FUNCTION_BLOCK CmdVentValves (* CAT Function Block Type *)
  (* Standard: 61499-2 *)
  (* Version 0.0, 6/8/2026, Schneider Electric, template *)
  PACKAGE SE.Nereda;
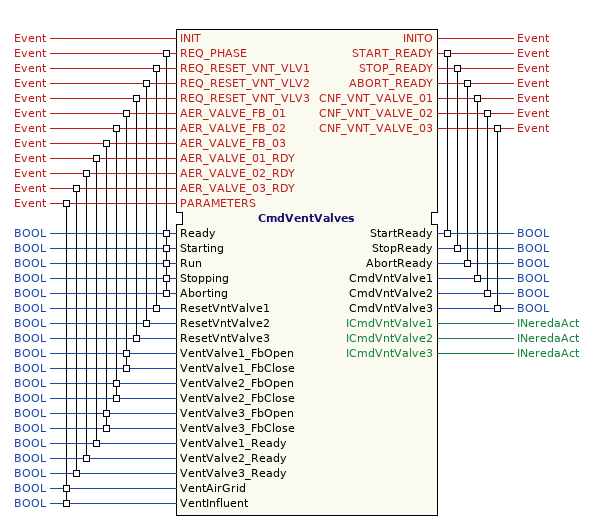
  EVENT_INPUT
    INIT;
    REQ_PHASE WITH Ready, Starting, Run, Stopping, Aborting;
    REQ_RESET_VNT_VLV1 WITH ResetVntValve1;
    REQ_RESET_VNT_VLV2 WITH ResetVntValve2;
    REQ_RESET_VNT_VLV3 WITH ResetVntValve3;
    AER_VALVE_FB_01 WITH VentValve1_FbOpen, VentValve1_FbClose;
    AER_VALVE_FB_02 WITH VentValve2_FbOpen, VentValve2_FbClose;
    AER_VALVE_FB_03 WITH VentValve3_FbOpen, VentValve3_FbClose;
    AER_VALVE_01_RDY WITH VentValve1_Ready;
    AER_VALVE_02_RDY WITH VentValve2_Ready;
    AER_VALVE_03_RDY WITH VentValve3_Ready;
    PARAMETERS WITH VentAirGrid, VentInfluent;
  END_EVENT
  EVENT_OUTPUT
    INITO;
    START_READY WITH StartReady;
    STOP_READY WITH StopReady;
    ABORT_READY WITH AbortReady;
    CNF_VNT_VALVE_01 WITH CmdVntValve1;
    CNF_VNT_VALVE_02 WITH CmdVntValve2;
    CNF_VNT_VALVE_03 WITH CmdVntValve3;
  END_EVENT
  VAR_INPUT
    Ready : BOOL;
    Starting : BOOL;
    Run : BOOL;
    Stopping : BOOL;
    Aborting : BOOL;
    ResetVntValve1 : BOOL;
    ResetVntValve2 : BOOL;
    ResetVntValve3 : BOOL;
    VentValve1_FbOpen : BOOL;
    VentValve1_FbClose : BOOL;
    VentValve2_FbOpen : BOOL;
    VentValve2_FbClose : BOOL;
    VentValve3_FbOpen : BOOL;
    VentValve3_FbClose : BOOL;
    VentValve1_Ready : BOOL;
    VentValve2_Ready : BOOL;
    VentValve3_Ready : BOOL;
    VentAirGrid : BOOL;
    VentInfluent : BOOL;
  END_VAR
  VAR_OUTPUT
    StartReady : BOOL;
    StopReady : BOOL;
    AbortReady : BOOL;
    CmdVntValve1 : BOOL;
    CmdVntValve2 : BOOL;
    CmdVntValve3 : BOOL;
  END_VAR
  PLUGS
    ICmdVntValve1 : INeredaAct;
    ICmdVntValve2 : INeredaAct;
    ICmdVntValve3 : INeredaAct;
  END_PLUGS
  (* 01 - FUNCTIONNAL INPUT INTERFACE *)
  (* 00 - INITIALIZATION *)
  (* 05 - LOGIC *)
  (* 06 - HMI INTERFACE *)
  (* 03 - FIELD INTERFACE *)
  (* 02 - FUNCTIONNAL OUTPUT INTERFACE *)
  (* Command Logic *)
  FBS
    IThis : CmdVentValves_HMI(QI := TRUE);
    CmdAerationValve1 : boolValueChanged;
    CmdAerationValve2 : boolValueChanged;
    FbOpenValve1 : DS_SELECTX_2536758B411A6CE51; {SET_ATTRIBUTE(Configuration.GenericFBType.InterfaceParams, Runtime.Standard#CNTX:=2;CNTY:=1;DI${CNTX,_,CNTY$}:BOOL)}
    FbCloseValve1 : DS_SELECTX_2536758B411A6CE51; {SET_ATTRIBUTE(Configuration.GenericFBType.InterfaceParams, Runtime.Standard#CNTX:=2;CNTY:=1;DI${CNTX,_,CNTY$}:BOOL)}
    FbOpenValve3 : DS_SELECTX_2536758B411A6CE51; {SET_ATTRIBUTE(Configuration.GenericFBType.InterfaceParams, Runtime.Standard#CNTX:=2;CNTY:=1;DI${CNTX,_,CNTY$}:BOOL)}
    FbCloseValve3 : DS_SELECTX_2536758B411A6CE51; {SET_ATTRIBUTE(Configuration.GenericFBType.InterfaceParams, Runtime.Standard#CNTX:=2;CNTY:=1;DI${CNTX,_,CNTY$}:BOOL)}
    FbReadyValve3 : DS_SELECTX_2536758B411A6CE51; {SET_ATTRIBUTE(Configuration.GenericFBType.InterfaceParams, Runtime.Standard#CNTX:=2;CNTY:=1;DI${CNTX,_,CNTY$}:BOOL)}
    FbReadyValve1 : DS_SELECTX_2536758B411A6CE51; {SET_ATTRIBUTE(Configuration.GenericFBType.InterfaceParams, Runtime.Standard#CNTX:=2;CNTY:=1;DI${CNTX,_,CNTY$}:BOOL)}
    FbOpenValve2 : DS_SELECTX_2536758B411A6CE51; {SET_ATTRIBUTE(Configuration.GenericFBType.InterfaceParams, Runtime.Standard#CNTX:=2;CNTY:=1;DI${CNTX,_,CNTY$}:BOOL)}
    FbCloseValve2 : DS_SELECTX_2536758B411A6CE51; {SET_ATTRIBUTE(Configuration.GenericFBType.InterfaceParams, Runtime.Standard#CNTX:=2;CNTY:=1;DI${CNTX,_,CNTY$}:BOOL)}
    FbReadyValve2 : DS_SELECTX_2536758B411A6CE51; {SET_ATTRIBUTE(Configuration.GenericFBType.InterfaceParams, Runtime.Standard#CNTX:=2;CNTY:=1;DI${CNTX,_,CNTY$}:BOOL)}
    CommandLogic : CmdVentValvesBasic;
    CmdAerationValve3 : boolValueChanged;
    Valve1Cmd : BOOL2INT;
    Valve2Cmd : BOOL2INT;
    Valve3Cmd : BOOL2INT;
  END_FBS
  EVENT_CONNECTIONS
    INIT TO IThis.3D5D26A512262747;
    IThis.5B84D78EC3FB5466 TO INITO;
    FbOpenValve1.CNF1 TO FbCloseValve1.REQ1;
    FbOpenValve1.CNF2 TO FbCloseValve1.REQ2;
    FbOpenValve3.CNF1 TO FbCloseValve3.REQ1;
    FbOpenValve3.CNF2 TO FbCloseValve3.REQ2;
    FbOpenValve2.CNF1 TO FbCloseValve2.REQ1;
    FbOpenValve2.CNF2 TO FbCloseValve2.REQ2;
    AER_VALVE_02_RDY TO FbReadyValve2.REQ2;
    AER_VALVE_01_RDY TO FbReadyValve1.REQ2;
    AER_VALVE_FB_02 TO FbOpenValve2.REQ2;
    AER_VALVE_FB_01 TO FbOpenValve1.REQ2;
    AER_VALVE_FB_03 TO FbOpenValve3.REQ2;
    AER_VALVE_03_RDY TO FbReadyValve3.REQ2;
    CommandLogic.2F06A37C5DC5770F TO IThis.FF79026EA8264D09;
    REQ_PHASE TO CommandLogic.0181C35002D51DB9;
    REQ_PHASE TO CommandLogic.7CF49D36E36F42BF;
    REQ_PHASE TO CommandLogic.270A548115E0D83C;
    REQ_PHASE TO CommandLogic.B01B36972B4703C3;
    REQ_PHASE TO CommandLogic.7D39C1849D7CD2AB;
    REQ_RESET_VNT_VLV1 TO ICmdVntValve1.37BBC1F841739733;
    REQ_RESET_VNT_VLV2 TO ICmdVntValve2.37BBC1F841739733;
    REQ_RESET_VNT_VLV3 TO ICmdVntValve3.37BBC1F841739733;
    PARAMETERS TO CommandLogic.PARAMETERS;
    FbCloseValve1.IND TO CommandLogic.VALVE_036_FB_STATE;
    FbCloseValve2.IND TO CommandLogic.VALVE_067_FB_STATE;
    FbCloseValve3.IND TO CommandLogic.D7181917E80A2E94;
    FbReadyValve1.IND TO CommandLogic.VALVE_036_AVAILABLE;
    FbReadyValve2.IND TO CommandLogic.VALVE_067_AVAILABLE;
    FbReadyValve3.IND TO CommandLogic.91B31299728D8852;
    CommandLogic.CNF_VALVE_36 TO CmdAerationValve1.REQ;
    CommandLogic.CNF_VALVE_67 TO CmdAerationValve2.REQ;
    CommandLogic.9605BD12A39689E0 TO CmdAerationValve3.REQ;
    CommandLogic.CNF_START_RDY TO START_READY;
    CommandLogic.CNF_STOP_RDY TO STOP_READY;
    CommandLogic.CNF_ABORT_RDY TO ABORT_READY;
    CmdAerationValve1.CHD TO Valve1Cmd.DD5870AA881150BB;
    CmdAerationValve2.CHD TO Valve2Cmd.DD5870AA881150BB;
    CmdAerationValve3.CHD TO Valve3Cmd.DD5870AA881150BB;
    Valve1Cmd.6FC99A5BD1C38561 TO ICmdVntValve1.0F1CDF9A9B4A227A;
    Valve2Cmd.6FC99A5BD1C38561 TO ICmdVntValve2.0F1CDF9A9B4A227A;
    Valve3Cmd.6FC99A5BD1C38561 TO ICmdVntValve3.0F1CDF9A9B4A227A;
    Valve1Cmd.6FC99A5BD1C38561 TO CNF_VNT_VALVE_01;
    Valve2Cmd.6FC99A5BD1C38561 TO CNF_VNT_VALVE_02;
    Valve3Cmd.6FC99A5BD1C38561 TO CNF_VNT_VALVE_03;
    ICmdVntValve1.9CD053F8408797ED TO FbOpenValve1.REQ1;
    ICmdVntValve1.CC753684FA882790 TO FbReadyValve1.REQ1;
    ICmdVntValve2.9CD053F8408797ED TO FbOpenValve2.REQ1;
    ICmdVntValve2.CC753684FA882790 TO FbReadyValve2.REQ1;
    ICmdVntValve3.9CD053F8408797ED TO FbOpenValve3.REQ1;
    ICmdVntValve3.CC753684FA882790 TO FbReadyValve3.REQ1;
  END_CONNECTIONS
  DATA_CONNECTIONS
    CmdAerationValve1.Output TO CmdVntValve1;
    CmdAerationValve2.Output TO CmdVntValve2;
    VentValve2_Ready TO FbReadyValve2.DI2_1;
    VentValve1_Ready TO FbReadyValve1.DI2_1;
    VentValve2_FbClose TO FbCloseValve2.DI2_1;
    VentValve2_FbOpen TO FbOpenValve2.DI2_1;
    VentValve1_FbClose TO FbCloseValve1.DI2_1;
    VentValve1_FbOpen TO FbOpenValve1.DI2_1;
    VentValve3_FbOpen TO FbOpenValve3.DI2_1;
    VentValve3_FbClose TO FbCloseValve3.DI2_1;
    VentValve3_Ready TO FbReadyValve3.DI2_1;
    CommandLogic.CB6518449836B6D0 TO IThis.73E7435EE8FD8D21;
    Ready TO CommandLogic.Ready;
    Starting TO CommandLogic.Starting;
    Run TO CommandLogic.Run;
    Stopping TO CommandLogic.Stopping;
    Aborting TO CommandLogic.Aborting;
    ResetVntValve1 TO ICmdVntValve1.EA28053F07575F36;
    ResetVntValve2 TO ICmdVntValve2.EA28053F07575F36;
    ResetVntValve3 TO ICmdVntValve3.EA28053F07575F36;
    VentAirGrid TO CommandLogic.AerationGrid;
    VentInfluent TO CommandLogic.InfluentGrid;
    CommandLogic.Valve036 TO CmdAerationValve1.Input;
    CommandLogic.Valve067 TO CmdAerationValve2.Input;
    CommandLogic.FA33A0628B344A4F TO CmdAerationValve3.Input;
    CommandLogic.StartReady TO StartReady;
    CommandLogic.StopReady TO StopReady;
    CommandLogic.AbortReady TO AbortReady;
    CmdAerationValve1.Output TO Valve1Cmd.4573FC8F228EB71D;
    CmdAerationValve2.Output TO Valve2Cmd.4573FC8F228EB71D;
    CmdAerationValve3.Output TO Valve3Cmd.4573FC8F228EB71D;
    Valve1Cmd.A6DEF5F9C27C1848 TO ICmdVntValve1.710D7FC54EE3F35A;
    Valve2Cmd.A6DEF5F9C27C1848 TO ICmdVntValve2.710D7FC54EE3F35A;
    Valve3Cmd.A6DEF5F9C27C1848 TO ICmdVntValve3.710D7FC54EE3F35A;
    CmdAerationValve3.Output TO CmdVntValve3;
    ICmdVntValve1.7F6CC7FEB9223DF3 TO FbOpenValve1.DI1_1;
    ICmdVntValve1.A8D6C4A1FDCCA991 TO FbCloseValve1.DI1_1;
    ICmdVntValve1.8A8A07EFCDA1443C TO FbReadyValve1.DI1_1;
    ICmdVntValve2.7F6CC7FEB9223DF3 TO FbOpenValve2.DI1_1;
    ICmdVntValve2.A8D6C4A1FDCCA991 TO FbCloseValve2.DI1_1;
    ICmdVntValve2.8A8A07EFCDA1443C TO FbReadyValve2.DI1_1;
    ICmdVntValve3.7F6CC7FEB9223DF3 TO FbOpenValve3.DI1_1;
    ICmdVntValve3.A8D6C4A1FDCCA991 TO FbCloseValve3.DI1_1;
    ICmdVntValve3.8A8A07EFCDA1443C TO FbReadyValve3.DI1_1;
    FbOpenValve1.OUT1 TO CommandLogic.Valve036_FbOpen;
    FbCloseValve1.OUT1 TO CommandLogic.Valve036_FbClose;
    FbOpenValve2.OUT1 TO CommandLogic.Valve067_FbOpen;
    FbCloseValve2.OUT1 TO CommandLogic.Valve067_FbClose;
    FbOpenValve3.OUT1 TO CommandLogic.0ADFB958CCA86E5C;
    FbCloseValve3.OUT1 TO CommandLogic.0DCCBC5ECDFE98C9;
    FbReadyValve1.OUT1 TO CommandLogic.Valve036_Availabe;
    FbReadyValve2.OUT1 TO CommandLogic.Valve067_Availabe;
    FbReadyValve3.OUT1 TO CommandLogic.B31B76F3A48A9DE5;
  END_CONNECTIONS
END_FUNCTION_BLOCK
